SUBAPPLICATION Uebung_122 (* Übung zu ISOBUS Name *)
  (* Standard: 61499-2; Description: Copyright (c) 2025 Meisterschulen am Ostbahnhof This program and the accompanying materials are made available under the terms of the Eclipse Public License 2.0 which is available at https://www.eclipse.org/legal/epl-2.0/ SPDX-License-Identifier: EPL-2.0 *)
  (* Version 1.0, 2023-10-23, Franz Höpfinger, Meisterschulen am Ostbahnhof *)
  IMPORT isobus::pgn::ISOUSERHOME_e;
  IMPORT isobus::pgn::ISO_CAN_NODE;
  IMPORT isobus::pgn::NAMEFIELD_T;
  IMPORT isobus::pgn::ISONETEVENT_T;
  IMPORT isobus::pgn::CF_INFO_T;
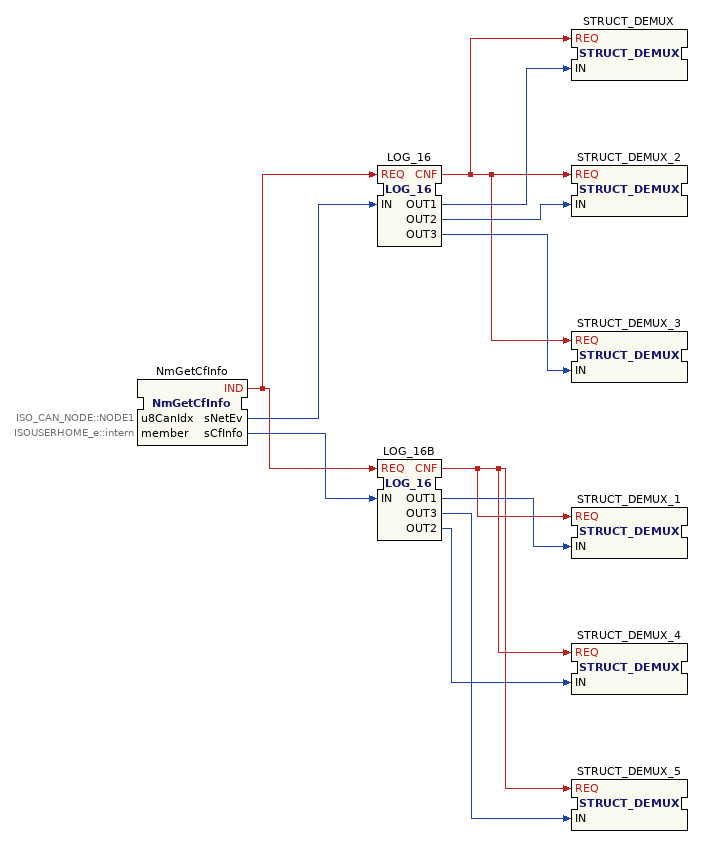
  FBS
    NmGetCfInfo : isobus::pgn::NmGetCfInfo(u8CanIdx := ISO_CAN_NODE::NODE1, member := ISOUSERHOME_e::intern);
    LOG_16 : eclipse4diac::utils::logging::LOG_16;
    LOG_16B : eclipse4diac::utils::logging::LOG_16;
    STRUCT_DEMUX : eclipse4diac::convert::STRUCT_DEMUX; {SET_ATTRIBUTE(StructuredType, isobus::pgn::ISONETEVENT_T)}
    STRUCT_DEMUX_1 : eclipse4diac::convert::STRUCT_DEMUX; {SET_ATTRIBUTE(StructuredType, isobus::pgn::CF_INFO_T)}
    STRUCT_DEMUX_2 : eclipse4diac::convert::STRUCT_DEMUX; {SET_ATTRIBUTE(StructuredType, isobus::pgn::ISONETEVENT_T)}
    STRUCT_DEMUX_3 : eclipse4diac::convert::STRUCT_DEMUX; {SET_ATTRIBUTE(StructuredType, isobus::pgn::ISONETEVENT_T)}
    STRUCT_DEMUX_4 : eclipse4diac::convert::STRUCT_DEMUX; {SET_ATTRIBUTE(StructuredType, isobus::pgn::CF_INFO_T)}
    STRUCT_DEMUX_5 : eclipse4diac::convert::STRUCT_DEMUX; {SET_ATTRIBUTE(StructuredType, isobus::pgn::CF_INFO_T)}
  END_FBS
  EVENT_CONNECTIONS
    NmGetCfInfo.IND TO LOG_16.REQ;
    NmGetCfInfo.IND TO LOG_16B.REQ;
    LOG_16.CNF TO STRUCT_DEMUX.REQ;
    LOG_16B.CNF TO STRUCT_DEMUX_1.REQ;
    LOG_16.CNF TO STRUCT_DEMUX_2.REQ;
    LOG_16.CNF TO STRUCT_DEMUX_3.REQ;
    LOG_16B.CNF TO STRUCT_DEMUX_4.REQ;
    LOG_16B.CNF TO STRUCT_DEMUX_5.REQ;
  END_CONNECTIONS
  DATA_CONNECTIONS
    NmGetCfInfo.sNetEv TO LOG_16.IN;
    NmGetCfInfo.sCfInfo TO LOG_16B.IN;
    LOG_16.OUT1 TO STRUCT_DEMUX.IN;
    LOG_16B.OUT1 TO STRUCT_DEMUX_1.IN;
    LOG_16.OUT2 TO STRUCT_DEMUX_2.IN;
    LOG_16.OUT3 TO STRUCT_DEMUX_3.IN;
    LOG_16B.OUT3 TO STRUCT_DEMUX_5.IN;
    LOG_16B.OUT2 TO STRUCT_DEMUX_4.IN;
  END_CONNECTIONS
END_SUBAPPLICATION
